{attribute 'linkalways'} 
{attribute 'no_explicit_call' := 'This FB is a CLASS and must be accessed using methods or properties'}
{attribute 'enable_dynamic_creation'}
FUNCTION_BLOCK FINAL MIN_SINT EXTENDS Node
VAR
	in1 : _SINT(0);
	in2 : _SINT(0);
	out : _SINT(0);
END_VAR

METHOD PUBLIC Clone : I_Node
VAR
	pNode : POINTER TO MIN_SINT;
END_VAR
pNode := __NEW(MIN_SINT);
Clone := pNode^;
END_METHOD

METHOD FB_init : BOOL
VAR_INPUT
	bInitRetains : BOOL; // if TRUE, the retain variables are initialized (warm start / cold start)
	bInCopyCode : BOOL;  // if TRUE, the instance afterwards gets moved into the copy code (online change)
END_VAR
AddInput('in1',THIS^.in1);
AddInput('in2',THIS^.in2);
AddOutput('out', THIS^.out);
END_METHOD

METHOD PROTECTED OnExecute
VAR
END_VAR
out.Value := MIN(in1.Value, in2.Value);
END_METHOD

END_FUNCTION_BLOCK

(* stored: Version 1.1.0.1, ProductVersion 3.1.4024.15
   POU MIN_SINT: Id {227cb5d4-319f-4f79-9fc2-77430f949e3d}, SpecialFunc None
   Folder Constructor: Id {c42c16ea-2d0e-4851-b9d9-5752263cbf1e}
   Method Clone: Id {bf7f0467-6357-4a48-bbe2-68d91efa7d35}
   Method FB_init: Id {6c1f3f02-3ace-4dce-9bd4-ac6d985489b9}
   Method OnExecute: Id {b28404c9-2acf-47d1-9afc-660ad47825b1} *)
